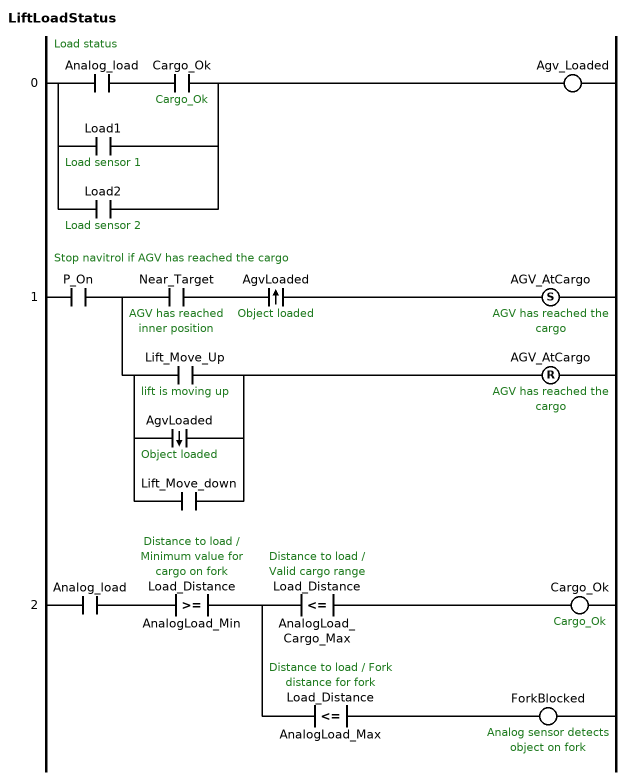
(* [picture p91: LiftLoadStatus, rungs 0-2] *)
(* Rung 0: Load status *)
Agv_Loaded := (Analog_load AND Cargo_Ok) OR Load1 OR Load2;
(* Rung 1: Stop navitrol if AGV has reached the cargo *)
_e1(CLK := AgvLoaded);
IF P_On AND Near_Target AND _e1.Q THEN AGV_AtCargo := TRUE; END_IF;
_e2(CLK := AgvLoaded);
IF P_On AND (Lift_Move_Up OR _e2.Q OR Lift_Move_down) THEN AGV_AtCargo := FALSE; END_IF;
(* Rung 2 *)
_p3 := Analog_load AND (Load_Distance >= AnalogLoad_Min);
Cargo_Ok := _p3 AND (Load_Distance <= AnalogLoad_Cargo_Max);
ForkBlocked := _p3 AND (Load_Distance <= AnalogLoad_Max);
END_FUNCTION_BLOCK

FUNCTION_BLOCK LiftAutoReset_FB
VAR
    DroppedFlag : BOOL;
END_VAR
VAR_INPUT
    Enable : BOOL;
    ControlMode : ControlLift;
    AgvLoaded : BOOL;
    Actuator_action : BOOL;
    Lift_height_actual : INT;
    Lift_height_empty : INT;
    Lift_heigt_loaded : INT;
    Dir_encoder : BOOL;
    UnloadDistance : DINT;
    M_per_rot : REAL;
    WheelEncPpr : REAL;
    ENC_position : DINT;
    ForkBlocked : BOOL;
END_VAR
VAR_OUTPUT
    ResetLift : BOOL;
    Reset_Lift_Busy : BOOL;
    Lift_Height_req_semiAuto : INT;
END_VAR
VAR_IN_OUT
    DroppedPosition : DINT;
    ResetDistance : DINT;
    ResetPosition : DINT;
END_VAR
VAR
    _e1 : F_TRIG;
    _p2 : BOOL;
    _e3 : R_TRIG;
END_VAR
(* ladder, written here as Structured Text *)

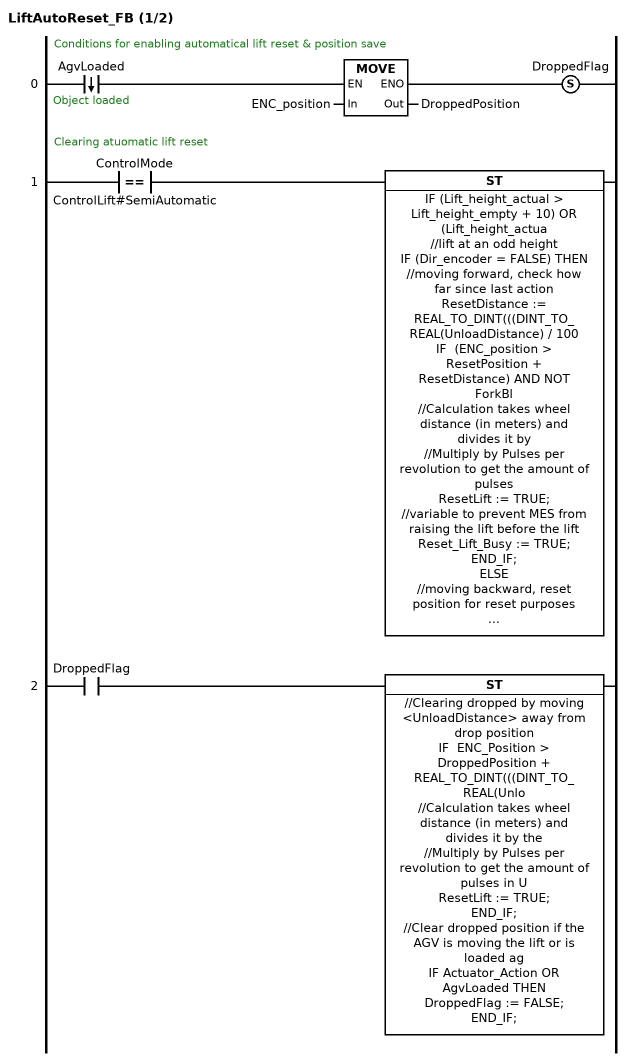
(* Rung 0: Conditions for enabling automatical lift reset & position save *)
_e1(CLK := AgvLoaded);
IF _e1.Q THEN
    DroppedPosition := ENC_position;
    DroppedFlag := TRUE;
END_IF;
(* Rung 1: Clearing atuomatic lift reset *)
IF ControlMode = ControlLift#SemiAutomatic THEN
    IF (Lift_height_actual > Lift_height_empty + 10) OR (Lift_height_actual < Lift_height_empty - 10) THEN
    	//lift at an odd height
    	IF (Dir_encoder = FALSE) THEN
    		//moving forward, check how far since last action
    		ResetDistance := REAL_TO_DINT(((DINT_TO_REAL(UnloadDistance) / 1000) / M_per_rot) * WheelEncPpr);
    		IF  (ENC_position > ResetPosition +  ResetDistance) AND NOT ForkBlocked THEN
    			//Calculation takes wheel distance (in meters) and divides it by the unload distance (in meters) to get the amount of wheel rotations in UnloadDistance. 
    			//Multiply by Pulses per revolution to get the amount of pulses in UnloadDistance.
    			ResetLift := TRUE;
    			//variable to prevent MES from raising the lift before the lift returned to normal
    			Reset_Lift_Busy := TRUE;
    		END_IF;
    	ELSE
    		//moving backward, reset position for reset purposes
    		ResetPosition := ENC_position;
    	END_IF;
    ELSE
    	//keep up with the current position
    	ResetPosition := ENC_position;
    END_IF;
END_IF;
(* Rung 2 *)
_p2 := DroppedFlag;
IF _p2 THEN
    //Clearing dropped by moving <UnloadDistance> away from drop position (and be sure fork is free)
    IF  ENC_Position > DroppedPosition +  REAL_TO_DINT(((DINT_TO_REAL(UnloadDistance) / 1000) / M_per_rot) * WheelEncPpr) AND NOT ForkBlocked THEN
    	//Calculation takes wheel distance (in meters) and divides it by the unload distance (in meters) to get the amount of wheel rotations in UnloadDistance. 
    	//Multiply by Pulses per revolution to get the amount of pulses in UnloadDistance.
    	ResetLift := TRUE;
    END_IF;
    //Clear dropped position if the AGV is moving the lift or is loaded again
    IF Actuator_Action OR AgvLoaded THEN
    	DroppedFlag := FALSE;
    END_IF;
END_IF;

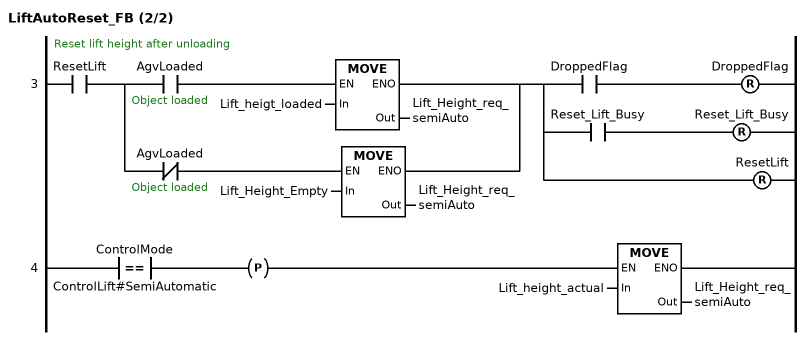
(* Rung 3: Reset lift height after unloading *)
IF ResetLift AND AgvLoaded THEN Lift_Height_req_semiAuto := Lift_heigt_loaded; END_IF;
IF ResetLift AND NOT AgvLoaded THEN Lift_Height_req_semiAuto := Lift_Height_Empty; END_IF;
IF ResetLift AND (AgvLoaded OR NOT AgvLoaded) AND DroppedFlag THEN DroppedFlag := FALSE; END_IF;
IF ResetLift AND (AgvLoaded OR NOT AgvLoaded) AND Reset_Lift_Busy THEN Reset_Lift_Busy := FALSE; END_IF;
IF ResetLift AND (AgvLoaded OR NOT AgvLoaded) THEN ResetLift := FALSE; END_IF;
(* Rung 4 *)
_e3(CLK := ControlMode = ControlLift#SemiAutomatic);
IF _e3.Q THEN Lift_Height_req_semiAuto := Lift_height_actual; END_IF;
END_FUNCTION_BLOCK

FUNCTION_BLOCK LiftCargoDrag_FB
VAR
    Difference_distance_drop : DINT;
    Difference_Pulses : REAL;
    Dropped_Flag : BOOL;
    Cargo_drag_TON : TON;
    Cargo_drag_flag : BOOL;
END_VAR
VAR_INPUT
    Enable : BOOL;
    Control_mode : ControlLift;
    Reset_flag : BOOL;
    Agv_loaded : BOOL;
    ENC_position : DINT;
    WheelEncPpr : REAL;
    M_per_Rot : REAL;
    Load_distance_real : REAL;
    Cargo_drag_PT : TIME;
END_VAR
VAR_OUTPUT
    Warning_cargo_drag : BOOL;
    Cargo_drag_ET : TIME;
END_VAR
VAR_IN_OUT
    Distance_traveled_in_m : REAL;
    Dropped_Position : DINT;
END_VAR
VAR_EXTERNAL
    AgvLoaded : BOOL;
END_VAR
VAR
    _e1 : F_TRIG;
    _e2 : R_TRIG;
END_VAR
(* ladder, written here as Structured Text *)

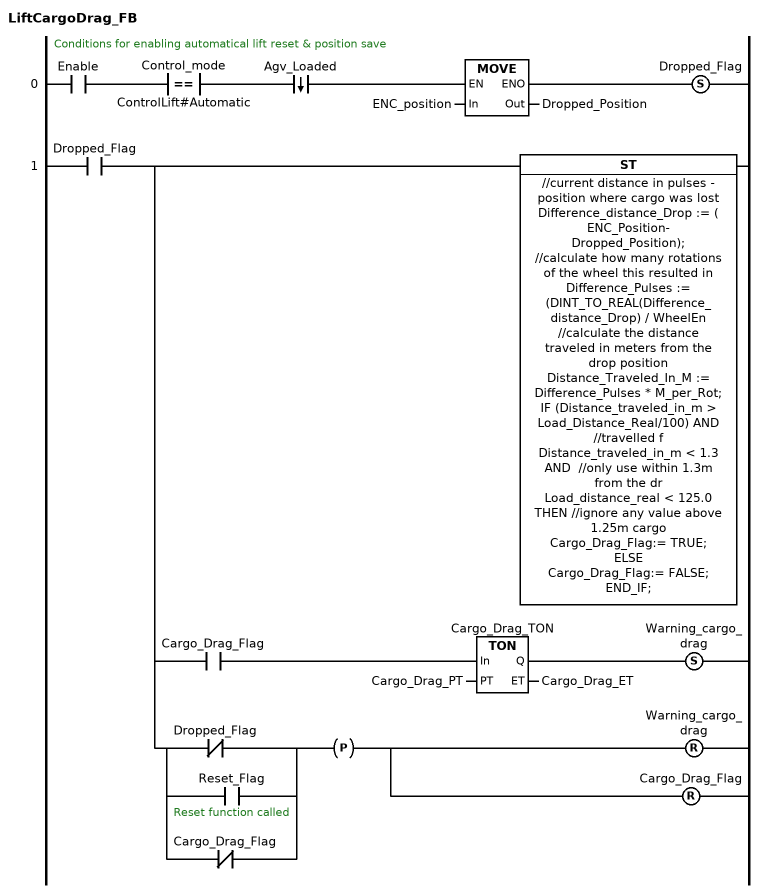
(* Rung 0: Conditions for enabling automatical lift reset & position save *)
_e1(CLK := Agv_Loaded);
IF Enable AND (Control_mode = ControlLift#Automatic) AND _e1.Q THEN
    Dropped_Position := ENC_position;
    Dropped_Flag := TRUE;
END_IF;
(* Rung 1 *)
IF Dropped_Flag THEN
    //current distance in pulses - position where cargo was lost
    Difference_distance_Drop := ( ENC_Position- Dropped_Position);
    //calculate how many rotations of the wheel this resulted in
    Difference_Pulses := (DINT_TO_REAL(Difference_distance_Drop) / WheelEncPpr);
    //calculate the distance traveled in meters from the drop position
    Distance_Traveled_In_M := Difference_Pulses * M_per_Rot;
    
    IF (Distance_traveled_in_m > Load_Distance_Real/100) AND //travelled further than the cargo?
    	Distance_traveled_in_m < 1.3 AND	//only use within 1.3m from the drop point
    	Load_distance_real < 125.0 THEN	//ignore any value above 1.25m cargo detection
    	Cargo_Drag_Flag:= TRUE;
    ELSE
    	Cargo_Drag_Flag:= FALSE;
    END_IF;
END_IF;
Cargo_Drag_TON(In := Dropped_Flag AND Cargo_Drag_Flag, PT := Cargo_Drag_PT, ET => Cargo_Drag_ET);
IF Cargo_Drag_TON.Q THEN Warning_cargo_drag := TRUE; END_IF;
_e2(CLK := Dropped_Flag AND (NOT Dropped_Flag OR Reset_Flag OR NOT Cargo_Drag_Flag));
IF _e2.Q THEN
    Warning_cargo_drag := FALSE;
    Cargo_Drag_Flag := FALSE;
END_IF;
END_FUNCTION_BLOCK

FUNCTION_BLOCK LiftHeavyLoadDetectionMax_FB
VAR_INPUT
    Enable : BOOL;
    Agv_heavy_Load_type_sensor : INT;  (* 0 = uses no sensor 1=digital sensor 2= analog sensor *)
    Heavy_weight_detection : BOOL;
    Max_weight : INT;
    Current_weight : INT;
END_VAR
VAR_OUTPUT
    Heavy_load : BOOL;
END_VAR
(* ladder, written here as Structured Text *)

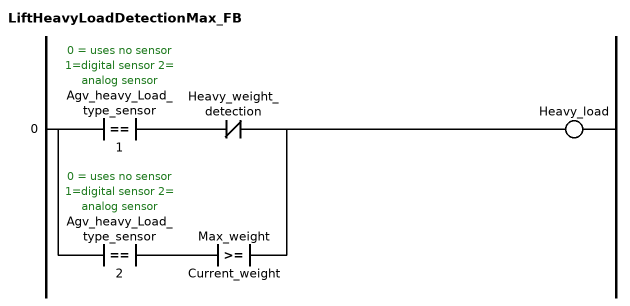
(* Rung 0 *)
Heavy_load := ((Agv_heavy_Load_type_sensor = 1) AND NOT Heavy_weight_detection) OR ((Agv_heavy_Load_type_sensor = 2) AND (Max_weight >= Current_weight));
END_FUNCTION_BLOCK

FUNCTION_BLOCK SendAckFatal
VAR
    DataReady : BOOL;  (* Data set ready for transmission *)
    TxBusy : BOOL;  (* Transmission in progress *)
    Data : Navitrol_AbortDrive_struct;
    SendDat : ARRAY[0..7] OF BYTE;  (* Data to send *)
    Messagesize : UINT;  (* Amount of bytes *)
    SendData : SktTCPSend;
END_VAR
VAR_INPUT
    Enable : BOOL;  (* Request to send *)
END_VAR
VAR_OUTPUT
    Done : BOOL;  (* Transmission done *)
END_VAR
VAR_INPUT
    Socket : _sSOCKET;  (* Navitrol socket *)
END_VAR
VAR_OUTPUT
    Error : BOOL;  (* Error during transmission *)
    ErrorID : WORD;  (* Error ID *)
END_VAR
VAR
    _e1 : R_TRIG;
    _p2 : BOOL;
    _p3 : BOOL;
    _e4 : R_TRIG;
END_VAR
(* ladder, written here as Structured Text *)

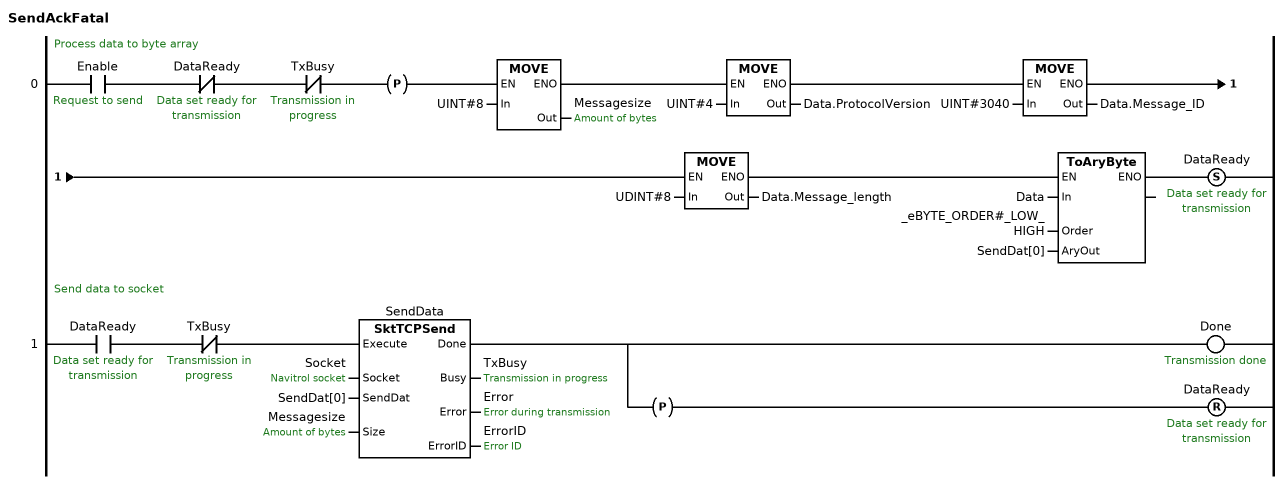
(* Rung 0: Process data to byte array *)
_e1(CLK := Enable AND NOT DataReady AND NOT TxBusy);
IF _e1.Q THEN
    Messagesize := UINT#8;
    Data.ProtocolVersion := UINT#4;
    Data.Message_ID := UINT#3040;
    Data.Message_length := UDINT#8;
    ToAryByte(In := Data, Order := _eBYTE_ORDER#_LOW_HIGH, AryOut := SendDat[0]);
    DataReady := TRUE;
END_IF;
(* Rung 1: Send data to socket *)
_p2 := DataReady AND NOT TxBusy;
SendData(Execute := _p2, Socket := Socket, SendDat := SendDat[0], Size := Messagesize, Busy => TxBusy, Error => Error, ErrorID => ErrorID);
_p3 := SendData.Done;
Done := _p3;
_e4(CLK := _p3);
IF _e4.Q THEN DataReady := FALSE; END_IF;
END_FUNCTION_BLOCK

FUNCTION_BLOCK WarningList
VAR
    WarningIndex : USINT;
END_VAR
VAR_OUTPUT
    OUT : BOOL;
END_VAR
VAR_INPUT
    IN : BOOL;
    i_BufferError : stBufferError;
    i_StoppedByOverhang : BOOL;
    ForkBlocked : BOOL;  (* Analog sensor detects object on fork *)
    Overhang_overruled : BOOL;
    FINS_enabled : BOOL;
    MES_Live : BOOL;
    StopByLowOpstacle : BOOL;
    SilentMode : BOOL;
END_VAR
VAR_EXTERNAL
    Scanner_Stop : BOOL;  (* object in safety field *)
    Warning_ActuatorTime : BOOL;  (* Lift action took too long *)
    Brake_release : BOOL;
    Manual_ControlModeLift : BOOL;
    Navitrol_status : Navitrol_Status_Struct;
    Scanner_Slowdown : BOOL;  (* object in slowdown field *)
    Scanner_Warning : BOOL;  (* object in outer field *)
    Warning_Cover_Open : BOOL;  (* One or more covers are not closed *)
    StopRequest : BOOL;
    AGV_Docking : BOOL;
    Warning_NoPallet : BOOL;  (* Cargo sensors did not detect load properly *)
    Warning_Lift_NOK : BOOL;  (* Lift sensor not in valid range *)
    Error_Navitrol : BOOL;  (* Navitrol reports an error *)
    WarningCount : USINT;  (* Amount of active warnings counter *)
    PLC_Warn_Array : array[0..4] of PLC_Warn_struct;
    Warning_TableLift_Without_load : BOOL;  (* Table has been ordered to rise without load present *)
    Warning_TableDrop_Without_Load : BOOL;  (* Table has been ordered to lower without load *)
    Warning_TableLoad_Lost : BOOL;  (* Lost tabel load while lift was high *)
    HMI_Warning1 : UINT;
    HMI_WarningText1 : INT;
    HMI_Warning2 : UINT;
    HMI_WarningText2 : INT;
    HMI_Warning3 : UINT;
    HMI_WarningText3 : INT;
    HMI_Warning4 : UINT;
    HMI_WarningText4 : INT;
    HMI_Warning5 : UINT;
    HMI_WarningText5 : INT;
    HMI_Input5 : BOOL;
    TCPReady : BOOL;
    AgvLoaded : BOOL;  (* Object loaded *)
    ClientConnected : BOOL;
    MQTT_enabled : BOOL;
    AGV_Docking_Lane : BOOL;
    HMI_Input12 : BOOL;
END_VAR
IF IN THEN		
		WarningCount := 0;

		IF AGV_Docking OR AGV_Docking_Lane then
			IF WarningCount < 5 THEN
				PLC_Warn_Array[WarningCount].WarnCode := 5101;
				PLC_Warn_Array[WarningCount].Description := 'Docking mode enabled';
				PLC_Warn_Array[WarningCount].HMI_id := 1;
				WarningCount := WarningCount + 1;
			END_IF;
		END_IF;

		IF Warning_TableLift_Without_load then
			IF WarningCount < 5 THEN
				PLC_Warn_Array[WarningCount].WarnCode := 5201;
				PLC_Warn_Array[WarningCount].Description := 'Pick without load';
				PLC_Warn_Array[WarningCount].HMI_id := 2;
				WarningCount := WarningCount + 1;
			END_IF;
		END_IF;

		IF Warning_TableDrop_Without_Load then
			IF WarningCount < 5 THEN
				PLC_Warn_Array[WarningCount].WarnCode := 5202;
				PLC_Warn_Array[WarningCount].Description := 'Drop without cargo';
				PLC_Warn_Array[WarningCount].HMI_id := 3;
				WarningCount := WarningCount + 1;
			END_IF;
		END_IF;

		IF Warning_TableLoad_Lost then
			IF WarningCount < 5 THEN
				PLC_Warn_Array[WarningCount].WarnCode := 5203;
				PLC_Warn_Array[WarningCount].Description := 'Lift has lost cargo';
				PLC_Warn_Array[WarningCount].HMI_id := 4;
				WarningCount := WarningCount + 1;
			END_IF;
		END_IF;

		IF Warning_ActuatorTime then
			IF WarningCount < 5 THEN
				PLC_Warn_Array[WarningCount].WarnCode := 5204;
				PLC_Warn_Array[WarningCount].Description := 'Actuator time exceeded';
				PLC_Warn_Array[WarningCount].HMI_id := 5;
				WarningCount := WarningCount + 1;
			END_IF;
		END_IF;

		IF MQTT_enabled AND Warning_NoPallet then
			IF WarningCount < 5 THEN
				PLC_Warn_Array[WarningCount].WarnCode := 5205;
				PLC_Warn_Array[WarningCount].Description := 'No cargo detected';
				PLC_Warn_Array[WarningCount].HMI_id := 6;
				WarningCount := WarningCount + 1;
			END_IF;
		END_IF;

		IF Warning_Lift_NOK then
			IF WarningCount < 5 THEN
				PLC_Warn_Array[WarningCount].WarnCode := 5206;
				PLC_Warn_Array[WarningCount].Description := 'Lift sensor out of range';
				PLC_Warn_Array[WarningCount].HMI_id := 7;
				WarningCount := WarningCount + 1;
			END_IF;
		END_IF;

		IF SilentMode then
			IF WarningCount < 5 THEN
				PLC_Warn_Array[WarningCount].WarnCode := 5301;
				PLC_Warn_Array[WarningCount].Description := 'Silent mode enabled';
				PLC_Warn_Array[WarningCount].HMI_id := 8;
				WarningCount := WarningCount + 1;
			END_IF;
		END_IF;

		IF Warning_Cover_Open then
			IF WarningCount < 5 THEN
				PLC_Warn_Array[WarningCount].WarnCode := 5401;
				PLC_Warn_Array[WarningCount].Description := 'Cover or door open';
				PLC_Warn_Array[WarningCount].HMI_id := 9;
				WarningCount := WarningCount + 1;
			END_IF;
		END_IF;

		IF WarningCount < 5 THEN
			IF Overhang_overruled then
				PLC_Warn_Array[WarningCount].WarnCode := 5403;
				PLC_Warn_Array[WarningCount].Description := 'Overhang overruled';
				PLC_Warn_Array[WarningCount].HMI_id := 11;
			ELSIF i_StoppedByOverhang then
				PLC_Warn_Array[WarningCount].WarnCode := 5402;
				PLC_Warn_Array[WarningCount].Description := 'Overhang detected';
				PLC_Warn_Array[WarningCount].HMI_id := 10;
			END_IF;
			WarningCount := WarningCount + 1;
		END_IF;


		IF Manual_ControlModeLift then
			IF WarningCount < 5 THEN
				PLC_Warn_Array[WarningCount].WarnCode := 5404;
				PLC_Warn_Array[WarningCount].Description := 'Manual mode active';
				PLC_Warn_Array[WarningCount].HMI_id := 12;
				WarningCount := WarningCount + 1;
			END_IF;
		END_IF;

		IF StopRequest then
			IF WarningCount < 5 THEN
				PLC_Warn_Array[WarningCount].WarnCode := 5405;
				PLC_Warn_Array[WarningCount].Description := 'Safety PLC stop request';
				PLC_Warn_Array[WarningCount].HMI_id := 13;
				WarningCount := WarningCount + 1;
			END_IF;
		END_IF;

		IF HMI_Input12 then
			IF WarningCount < 5 THEN
				PLC_Warn_Array[WarningCount].WarnCode := 5406;
				PLC_Warn_Array[WarningCount].Description := 'Operator deleted action';
				PLC_Warn_Array[WarningCount].HMI_id := 14;
				WarningCount := WarningCount + 1;
			END_IF;
		END_IF;

		IF Scanner_Warning & Scanner_Slowdown & NOT Scanner_Stop then
			IF WarningCount < 5 THEN
				PLC_Warn_Array[WarningCount].WarnCode := 5501;
				PLC_Warn_Array[WarningCount].Description := 'Object in stop field';
				PLC_Warn_Array[WarningCount].HMI_id := 15;
				WarningCount := WarningCount + 1;
			END_IF;
		END_IF;

		IF Error_Navitrol & (Navitrol_status.Pos_Conf > 30) then
			IF WarningCount < 5 THEN
				PLC_Warn_Array[WarningCount].WarnCode := 5602;
				PLC_Warn_Array[WarningCount].Description := 'Navigation in error';
				PLC_Warn_Array[WarningCount].HMI_id := 17;
				WarningCount := WarningCount + 1;
			END_IF;
		END_IF;

		IF Error_Navitrol & (Navitrol_status.Pos_Conf < 30) then
			IF WarningCount < 5 THEN
				PLC_Warn_Array[WarningCount].WarnCode := 5603;
				PLC_Warn_Array[WarningCount].Description := 'Navigation is lost';
				PLC_Warn_Array[WarningCount].HMI_id := 18;
				WarningCount := WarningCount + 1;
			END_IF;
		END_IF;

		IF p_off then
			IF WarningCount < 5 THEN
				PLC_Warn_Array[WarningCount].WarnCode := 5207;
				PLC_Warn_Array[WarningCount].Description := 'Pallet override active';
				PLC_Warn_Array[WarningCount].HMI_id := 19;
				WarningCount := WarningCount + 1;
			END_IF;
		END_IF;

		IF ForkBlocked AND NOT AgvLoaded then
			IF WarningCount < 5 THEN
				PLC_Warn_Array[WarningCount].WarnCode := 5209;
				PLC_Warn_Array[WarningCount].Description := 'Cargo location invalid';
				PLC_Warn_Array[WarningCount].HMI_id := 21;
				WarningCount := WarningCount + 1;
			END_IF;
		END_IF;

		IF Brake_release then
			IF WarningCount < 5 THEN
				PLC_Warn_Array[WarningCount].WarnCode := 5407;
				PLC_Warn_Array[WarningCount].Description := 'Brakes released';
				PLC_Warn_Array[WarningCount].HMI_id := 22;
				WarningCount := WarningCount + 1;
			END_IF;
		END_IF;

		IF HMI_Input5 then
			IF WarningCount < 5 THEN
				PLC_Warn_Array[WarningCount].WarnCode := 5408;
				PLC_Warn_Array[WarningCount].Description := 'Lift action overruled';
				PLC_Warn_Array[WarningCount].HMI_id := 23;
				WarningCount := WarningCount + 1;
			END_IF;
		END_IF;

		//communication warnings
		IF (NOT TCPReady) THEN
			IF WarningCount < 5 THEN
				PLC_Warn_Array[WarningCount].WarnCode := 5701;
				PLC_Warn_Array[WarningCount].Description := 'Navitrol offline';
				PLC_Warn_Array[WarningCount].HMI_id := 24;
				WarningCount := WarningCount + 1;
			END_IF;
		END_IF;

		IF (FINS_enabled AND NOT MES_Live) THEN
			IF WarningCount < 5 THEN
				PLC_Warn_Array[WarningCount].WarnCode := 5702;
				PLC_Warn_Array[WarningCount].Description := 'FINS timeout to MES';
				PLC_Warn_Array[WarningCount].HMI_id := 25;
				WarningCount := WarningCount + 1;
			END_IF;
		END_IF;

		IF (MQTT_enabled AND NOT ClientConnected) THEN
			IF WarningCount < 5 THEN
				PLC_Warn_Array[WarningCount].WarnCode := 5703;
				PLC_Warn_Array[WarningCount].Description := 'Mqtt broker offline';
				PLC_Warn_Array[WarningCount].HMI_id := 26;
				WarningCount := WarningCount + 1;
			END_IF;
		END_IF;

		(*IF  then
			IF WarningCount < 5 THEN
				PLC_Warn_Array[WarningCount].WarnCode := 5405;
				PLC_Warn_Array[WarningCount].Description := 'AGV in stopzone';
				PLC_Warn_Array[WarningCount].HMI_id := 27;
				WarningCount := WarningCount + 1;
			END_IF;
		END_IF;

		IF  then
			IF WarningCount < 5 THEN
				PLC_Warn_Array[WarningCount].WarnCode := 5210;
				PLC_Warn_Array[WarningCount].Description := 'Pallet stack height detection active';
				PLC_Warn_Array[WarningCount].HMI_id := 28;
				WarningCount := WarningCount + 1;
			END_IF;
		END_IF;

		IF  then
			IF WarningCount < 5 THEN
				PLC_Warn_Array[WarningCount].WarnCode := 5211;
				PLC_Warn_Array[WarningCount].Description := 'Too many pallets detect.';
				PLC_Warn_Array[WarningCount].HMI_id := 29;
				WarningCount := WarningCount + 1;
			END_IF;
		END_IF;
		*)

		IF StopByLowOpstacle then
			IF WarningCount < 5 THEN
				PLC_Warn_Array[WarningCount].WarnCode := 5409;
				PLC_Warn_Array[WarningCount].Description := 'Low sensor detec object';
				PLC_Warn_Array[WarningCount].HMI_id := 30;
				WarningCount := WarningCount + 1;
			END_IF;
		END_IF;
		
		IF P_Off THEN
			IF WarningCount < 5 THEN
				PLC_Warn_Array[WarningCount].WarnCode := 5411;
				PLC_Warn_Array[WarningCount].Description := 'Lane sensor out of range';
				PLC_Warn_Array[WarningCount].HMI_id := 31;
				WarningCount := WarningCount + 1;
			END_IF;
		END_IF;

		IF i_BufferError.LiftHeight THEN
			IF WarningCount < 5 THEN
				PLC_Warn_Array[WarningCount].WarnCode := 5412;
				PLC_Warn_Array[WarningCount].Description := 'Too low lift height lane';
				PLC_Warn_Array[WarningCount].HMI_id := 32;
				WarningCount := WarningCount + 1;
			END_IF;
		END_IF;
		
		IF i_BufferError.CargoSensorBWIRE THEN
			IF WarningCount < 5 THEN
				PLC_Warn_Array[WarningCount].WarnCode := 5413;
				PLC_Warn_Array[WarningCount].Description := 'Cargo sensor broke wire';
				PLC_Warn_Array[WarningCount].HMI_id := 33;
				WarningCount := WarningCount + 1;
			END_IF;
		END_IF;

		IF (WarningCount < 5) THEN
			PLC_Warn_Array[4].WarnCode := 0;
			PLC_Warn_Array[4].Description := '                        ';
			PLC_Warn_Array[4].HMI_id := 0;
		END_IF;
		IF (WarningCount < 4) THEN
			PLC_Warn_Array[3].WarnCode := 0;
			PLC_Warn_Array[3].Description := '                        ';
			PLC_Warn_Array[3].HMI_id := 0;
		END_IF;
		IF (WarningCount < 3) THEN
			PLC_Warn_Array[2].WarnCode := 0;
			PLC_Warn_Array[2].Description := '                        ';
			PLC_Warn_Array[2].HMI_id := 0;
		END_IF;
		IF (WarningCount < 2) THEN
			PLC_Warn_Array[1].WarnCode := 0;
			PLC_Warn_Array[1].Description := '                        ';
			PLC_Warn_Array[1].HMI_id := 0;
		END_IF;
		IF (WarningCount < 1) THEN
			//no warnings active
			PLC_Warn_Array[0].WarnCode := 0;
			PLC_Warn_Array[0].Description := '                        ';
			PLC_Warn_Array[0].HMI_id := 0;
		END_IF;

		//Handle the error strings
		FOR WarningIndex := 0 to 4 DO
			PLC_Warn_Array[WarningIndex].ActualChars := uint_to_byte(LEN(PLC_Warn_Array[WarningIndex].Description));
			PLC_Warn_Array[WarningIndex].ZeroFill := int_to_byte(BYTE_TO_INT(PLC_Warn_Array[WarningIndex].DescrLength) -BYTE_TO_INT(PLC_Warn_Array[WarningIndex].ActualChars));
		END_FOR;

		//HMI_WarningText1 := '                        ';
		//HMI_WarningText2 := '                        ';
		//HMI_WarningText3 := '                        ';
		//HMI_WarningText4 := '                        ';
		//HMI_WarningText5 := '                        ';

		HMI_Warning1 := PLC_Warn_Array[0].WarnCode;
		HMI_WarningText1 := BYTE_TO_INT(PLC_Warn_Array[0].HMI_id);
		HMI_Warning2 := PLC_Warn_Array[1].WarnCode;
		HMI_WarningText2 :=  BYTE_TO_INT(PLC_Warn_Array[1].HMI_id);
		HMI_Warning3 := PLC_Warn_Array[2].WarnCode;
		HMI_WarningText3 :=  BYTE_TO_INT(PLC_Warn_Array[2].HMI_id);
		HMI_Warning4 := PLC_Warn_Array[3].WarnCode;
		HMI_WarningText4 :=  BYTE_TO_INT(PLC_Warn_Array[3].HMI_id);
		HMI_Warning5 := PLC_Warn_Array[4].WarnCode;
		HMI_WarningText5 :=  BYTE_TO_INT(PLC_Warn_Array[4].HMI_id);
END_IF;
END_FUNCTION_BLOCK

FUNCTION_BLOCK Bufferlane_FB
VAR
    STANDSTILL_CARGO_DIST_MIN : REAL := 970;  (* Minimum value cargo should be *)
    DistSensor : stAnalogSensor;
    LoadSwitchDelay1 : TOF;
    NAVITROL_BUFFERLANE_FIRST : REAL := 1;  (* AGV in bufferlane *)
    BUFFERLANE_PICK : INT := 1;  (* MES defined action 1 *)
    BUFFERLANE_DROP : INT := 2;  (* MES defined action 2 *)
    BUFFERLANE_DROP_HEIGHT : INT := 295;  (* Drop height in bufferlane, customer Alpma *)
    HoldOnPosition : BOOL;  (* Keep AGV on position *)
    BUFFERLANE_PICK_HEIGHT : INT := 460;  (* Pick height in bufferlane, customer Alpma *)
    PICKING_ACTION : INT := 40;  (* Enum values picking *)
    DROPPING_ACTION : INT := 40;  (* Enum values dropping *)
    TARGET_REACHED : UINT := 1;
    ENTER_LANE_LIFT_MARGE : INT := 10;
    NAVITROL_BUFFERLANE_OUT : REAL := 4;
    DIST_TO_TARGET_MIN : REAL := 0.2;  (* AGV does stop at target instead sensor *)
    SP_SLOW : INT;
    SP_STOP : INT;
    ANALOG_LANE_SENSOR : INT := 1;  (* Analog sensor to stop AGV *)
END_VAR
VAR_INPUT
    ENABLE : BOOL;
    CNTRL : stControl;
    i_LaneStateMES : Lane_state_MES;
    i_SensorType : INT;
    i_BufferLaneSensorDistance : INT;
    i_Load_Distance : REAL;
    i_LiftReqAuto : INT;
    i_ClampSTS : BOOL;
    i_Lift_Height : INT;  (* Calculated lift height *)
    i_ReadyToClamp : BOOL;  (* Calculated lift height *)
    i_Lift_Mode : ControlLift;  (* Lift control mode *)
END_VAR
VAR_OUTPUT
    STOP_POS : BOOL;  (* AGV stopped by used distance and cargo sensor *)
    SPD_LIM : BOOL;  (* AGV gets limited in speed *)
    STATUS : stBufferlaneStatus;
    ErrType : stBufferError;
    ERROR : BOOL;
END_VAR
VAR_EXTERNAL
    Load_Distance : INT;
    Manual_Navitrol : BOOL;
    Navitrol_ProductionStatus : Navitrol_ProductionData_struct;
    Navitrol_DriveInfo : Navitrol_Status_DriveorderInfo_sec_struct;
    Navitrol_DistanceInfo : Navitrol_Status_DistanceToTarget_sec_struct;
    Standstill : BOOL;
    ClampAttached : BOOL;
    Scan3_Stop : BOOL;
    Scan3_Warn : BOOL;
    ActuatorAction : BOOL;
    RequestDriveReady : BOOL;
END_VAR
VAR
    _e1 : F_TRIG;
    _e2 : F_TRIG;
    _e3 : R_TRIG;
    _e4 : R_TRIG;
    _e5 : R_TRIG;
    _e6 : R_TRIG;
    _e7 : R_TRIG;
    _e8 : R_TRIG;
    _e9 : F_TRIG;
END_VAR
(* ladder, written here as Structured Text *)

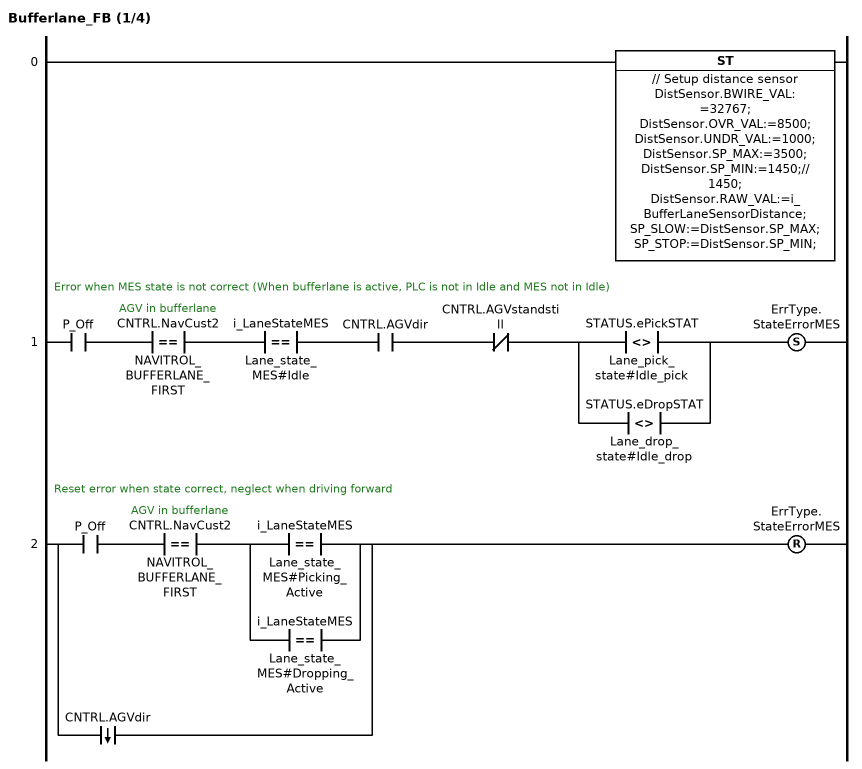
(* Rung 0 *)
// Setup distance sensor

DistSensor.BWIRE_VAL:=32767;
DistSensor.OVR_VAL:=8500;
DistSensor.UNDR_VAL:=1000;
DistSensor.SP_MAX:=3500;
DistSensor.SP_MIN:=1450;//1450;
DistSensor.RAW_VAL:=i_BufferLaneSensorDistance;

SP_SLOW:=DistSensor.SP_MAX;
SP_STOP:=DistSensor.SP_MIN;
(* Rung 1: Error when MES state is not correct (When bufferlane is active, PLC is not in Idle and MES not in Idle) *)
IF P_Off AND (CNTRL.NavCust2 = NAVITROL_BUFFERLANE_FIRST) AND (i_LaneStateMES = Lane_state_MES#Idle) AND CNTRL.AGVdir AND NOT CNTRL.AGVstandstill AND ((STATUS.ePickSTAT <> Lane_pick_state#Idle_pick) OR (STATUS.eDropSTAT <> Lane_drop_state#Idle_drop)) THEN
    ErrType.StateErrorMES := TRUE;
END_IF;
(* Rung 2: Reset error when state correct, neglect when driving forward *)
_e1(CLK := CNTRL.AGVdir);
IF (P_Off AND (CNTRL.NavCust2 = NAVITROL_BUFFERLANE_FIRST) AND ((i_LaneStateMES = Lane_state_MES#Picking_Active) OR (i_LaneStateMES = Lane_state_MES#Dropping_Active))) OR _e1.Q THEN
    ErrType.StateErrorMES := FALSE;
END_IF;

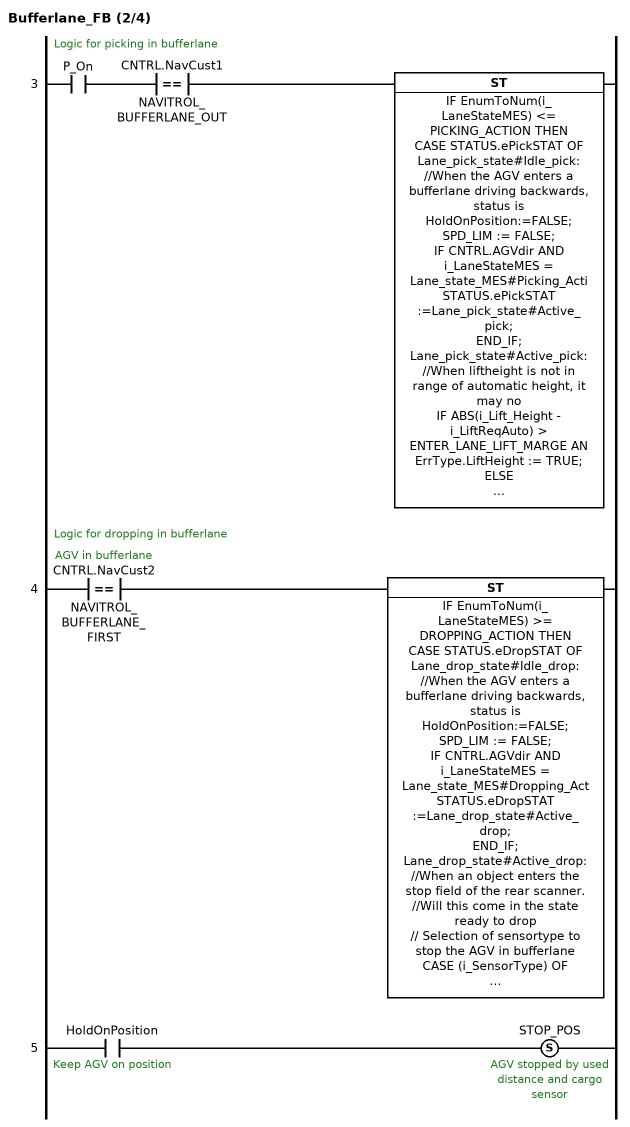
(* Rung 3: Logic for picking in bufferlane *)
IF P_On AND (CNTRL.NavCust1 = NAVITROL_BUFFERLANE_OUT) THEN
    IF EnumToNum(i_LaneStateMES) <= PICKING_ACTION THEN	
    	CASE STATUS.ePickSTAT OF
    		Lane_pick_state#Idle_pick:
    			//When the AGV enters a bufferlane driving backwards, status is active pick
    			HoldOnPosition:=FALSE;
    			SPD_LIM := FALSE;
    			IF CNTRL.AGVdir AND i_LaneStateMES = Lane_state_MES#Picking_Active THEN 
    				STATUS.ePickSTAT :=Lane_pick_state#Active_pick;
    			END_IF;
    
    		Lane_pick_state#Active_pick:
    			//When liftheight is not in range of automatic height, it may not drive automatically in lane!
    			IF ABS(i_Lift_Height - i_LiftReqAuto) > ENTER_LANE_LIFT_MARGE AND CNTRL.AGVdir AND CNTRL.NavInProduction  = 1 THEN
    				ErrType.LiftHeight := TRUE;
    			ELSE
    				ErrType.LiftHeight := FALSE;
    			END_IF;
    			
    			// Selection of sensortype to stop the AGV in bufferlane
    			CASE (i_SensorType) OF
    				1:
    					//Analog has max setpoint for slowdown and min setpoint for stopping AGV
    					IF DistSensor.RAW_VAL < SP_SLOW THEN
    						SPD_LIM := TRUE;
    					END_IF;
    					IF DistSensor.RAW_VAL < SP_STOP AND CNTRL.AGVdir THEN
    						HoldOnPosition := TRUE;
    						IF CNTRL.AGVstandstill AND i_LaneStateMES = Lane_state_MES#Picking_Active THEN
    							STATUS.ePickSTAT := Ready_to_lower_lift_pick;
    						END_IF;
    					END_IF;
    				
    				//AGV stopts already when safety scanner sees an object in stopfield
    				2:
    					IF Scan3_Stop THEN
    						IF CNTRL.AGVstandstill AND i_LaneStateMES = Lane_state_MES#Picking_Active THEN
    							STATUS.ePickSTAT := Ready_to_lower_lift_pick;
    						END_IF;
    					END_IF;				
    			END_CASE;
    			
    		
    		Lane_pick_state#Ready_to_lower_lift_pick:
    			// HoldOnPosition while lowering lift
    			HoldOnPosition := ActuatorAction;
    		
    			//When the lift is lowered, AGV can drive with forks under load
    			IF i_LaneStateMES = Lane_state_MES#Picking_Drive_In THEN
    				HoldOnPosition := FALSE;
    			END_IF;
    			//AGV does not stop on cargo sensor, but symbolic point if distance is less than DIST_TO_TARGET_MIN
    			IF Navitrol_DistanceInfo.DistanceToTarget <= DIST_TO_TARGET_MIN THEN
    				IF NOT i_ReadyToClamp AND CNTRL.AGVstandstill THEN
    					STATUS.ePickSTAT := Ready_to_pick;
    				END_IF;
    			ELSE
    			//Otherwise AGV stops when it is loaded
    				IF CNTRL.AGVloaded THEN
    					HoldOnPosition:=TRUE;
    					IF NOT i_ReadyToClamp AND CNTRL.AGVstandstill THEN
    						STATUS.ePickSTAT := Ready_to_pick;
    					END_IF;
    				END_IF;
    			END_IF;
    			
    		Lane_pick_state#Ready_to_pick:
    			//When the AGV has picked the cargo, it will be reversed by the MES application.
    			//From that moment on, the state is changed to idle.
    			IF i_LaneStateMES = Lane_state_MES#Picking_Finished THEN
    				IF ClampAttached AND i_ClampSTS THEN
    					STATUS.ePickSTAT := Idle_pick;
    				ELSIF NOT ClampAttached THEN
    					STATUS.ePickSTAT := Idle_pick;
    				END_IF;
    			END_IF;
    	END_CASE;
    
    	//When the AGV drives out the lane-picking lane, the lanepick state is written to idle.
    	IF NOT CNTRL.AGVdir AND NOT CNTRL.AGVstandstill THEN
    		STATUS.ePickSTAT := Idle_pick;
    	END_IF;
    END_IF;
END_IF;
(* Rung 4: Logic for dropping in bufferlane *)
IF CNTRL.NavCust2 = NAVITROL_BUFFERLANE_FIRST THEN
    IF EnumToNum(i_LaneStateMES) >= DROPPING_ACTION THEN	
    	CASE STATUS.eDropSTAT OF
    		Lane_drop_state#Idle_drop:
    			//When the AGV enters a bufferlane driving backwards, status is active drop
    			HoldOnPosition:=FALSE;
    			SPD_LIM := FALSE;
    			IF CNTRL.AGVdir AND i_LaneStateMES = Lane_state_MES#Dropping_Active THEN
    				STATUS.eDropSTAT :=Lane_drop_state#Active_drop;
    			END_IF;
    
    		Lane_drop_state#Active_drop:
    			//When an object enters the stop field of the rear scanner.
    			//Will this come in the state ready to drop	
    			
    			// Selection of sensortype to stop the AGV in bufferlane
    			CASE (i_SensorType) OF
    				1:
    					//Analog has max setpoint for slowdown and min setpoint for stopping AGV
    					IF DistSensor.RAW_VAL < SP_SLOW AND DistSensor.RAW_VAL > SP_STOP THEN
    						SPD_LIM := TRUE;
    					END_IF;
    					IF DistSensor.RAW_VAL < SP_STOP AND DistSensor.RAW_VAL > DistSensor.UNDR_VAL AND CNTRL.AGVdir  THEN
    						HoldOnPosition:=TRUE;
    						IF CNTRL.AGVstandstill AND i_LaneStateMES = Lane_state_MES#Dropping_Active THEN
    							STATUS.eDropSTAT := Ready_to_drop;
    						END_IF;	
    					END_IF;	
    				2:
    					//AGV stopts already when safety scanner sees an object in stopfield
    					IF Scan3_Stop AND Standstill THEN						 
    						IF CNTRL.AGVstandstill AND i_LaneStateMES = Lane_state_MES#Dropping_Active THEN
    							STATUS.eDropSTAT := Ready_to_drop;
    						END_IF;
    					END_IF;
    			END_CASE;
    			
    			IF i_LaneStateMES = Lane_state_MES#Dropping THEN
    					STATUS.eDropSTAT := Ready_to_drop;
    			END_IF;
    
    		Lane_drop_state#Ready_to_drop:
    			//When the AGV has dropped the pallet, it will be reversed by the MES application.
    			//And when the AGV has moved backwards enough, the lift is sent upwards.
    			//From that moment on, the state is changed to finshed.	
    			
    			// HoldOnPosition while lowering lift
    			HoldOnPosition := ActuatorAction;
    			RequestDriveReady:=TRUE;
    			
    			IF CNTRL.AGVstandstill AND i_LaneStateMES = Lane_state_MES#Dropping_Finished THEN
    				STATUS.eDropSTAT := Idle_drop;
    			END_IF;
    	END_CASE;
    
    	//When the agv is not in a lane-dropping lane.
    	//The lanedrop state is written to idle.
    	IF NOT CNTRL.AGVdir AND NOT CNTRL.AGVstandstill THEN
    		STATUS.eDropSTAT := Idle_drop;
    	END_IF;
    END_IF;
END_IF;
(* Rung 5 *)
IF HoldOnPosition THEN STOP_POS := TRUE; END_IF;

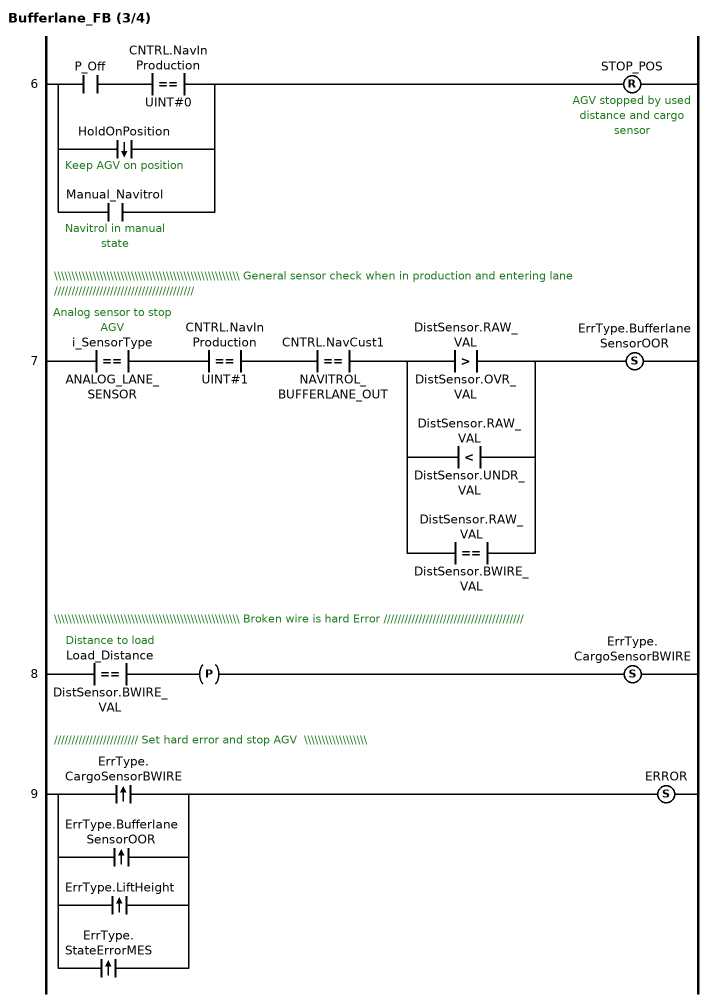
(* Rung 6 *)
_e2(CLK := HoldOnPosition);
IF (P_Off AND (CNTRL.NavInProduction = UINT#0)) OR _e2.Q OR Manual_Navitrol THEN
    STOP_POS := FALSE;
END_IF;
(* Rung 7: \\\\\\\\\\\\\\\\\\\\\\\\\\\\\\\\\\\\\\\\\\\\\\\\\\\\\ General sensor check when in production and entering lane //////////////////////////////////////// *)
IF (i_SensorType = ANALOG_LANE_SENSOR) AND (CNTRL.NavInProduction = UINT#1) AND (CNTRL.NavCust1 = NAVITROL_BUFFERLANE_OUT) AND ((DistSensor.RAW_VAL > DistSensor.OVR_VAL) OR (DistSensor.RAW_VAL < DistSensor.UNDR_VAL) OR (DistSensor.RAW_VAL = DistSensor.BWIRE_VAL)) THEN
    ErrType.BufferlaneSensorOOR := TRUE;
END_IF;
(* Rung 8: \\\\\\\\\\\\\\\\\\\\\\\\\\\\\\\\\\\\\\\\\\\\\\\\\\\\\ Broken wire is hard Error //////////////////////////////////////// *)
_e3(CLK := Load_Distance = DistSensor.BWIRE_VAL);
IF _e3.Q THEN ErrType.CargoSensorBWIRE := TRUE; END_IF;
(* Rung 9: //////////////////////// Set hard error and stop AGV  \\\\\\\\\\\\\\\\\\ *)
_e4(CLK := ErrType.CargoSensorBWIRE);
_e5(CLK := ErrType.BufferlaneSensorOOR);
_e6(CLK := ErrType.LiftHeight);
_e7(CLK := ErrType.StateErrorMES);
IF _e4.Q OR _e5.Q OR _e6.Q OR _e7.Q THEN ERROR := TRUE; END_IF;

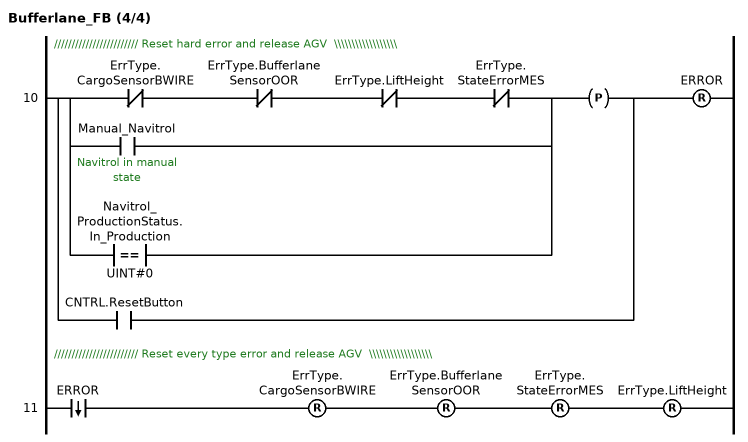
(* Rung 10: //////////////////////// Reset hard error and release AGV  \\\\\\\\\\\\\\\\\\ *)
_e8(CLK := (NOT ErrType.CargoSensorBWIRE AND NOT ErrType.BufferlaneSensorOOR AND NOT ErrType.LiftHeight AND NOT ErrType.StateErrorMES) OR Manual_Navitrol OR (Navitrol_ProductionStatus.In_Production = UINT#0));
IF _e8.Q OR CNTRL.ResetButton THEN ERROR := FALSE; END_IF;
(* Rung 11: //////////////////////// Reset every type error and release AGV  \\\\\\\\\\\\\\\\\\ *)
_e9(CLK := ERROR);
IF _e9.Q THEN
    ErrType.CargoSensorBWIRE := FALSE;
    ErrType.BufferlaneSensorOOR := FALSE;
    ErrType.StateErrorMES := FALSE;
    ErrType.LiftHeight := FALSE;
END_IF;
END_FUNCTION_BLOCK

FUNCTION_BLOCK ErrorList_FB
VAR_INPUT
    IN : BOOL;
END_VAR
VAR_OUTPUT
    OUT : BOOL;
END_VAR
VAR_EXTERNAL
    ErrorCount : USINT;
    Motor_Ok : BOOL;
    PLC_Error_Array : array[0..4] of PLC_Error_struct;
    Estop_Channel1 : BOOL;
    Error_Fork_Object : BOOL;
    Docking_error : BOOL;
    SpeedError : BOOL;
    Pump_Ok : BOOL;
    Estop_Out : BOOL;
    Scanner_Warning : BOOL;
    Scanner_Slowdown : BOOL;
    Scanner_Stop : BOOL;
    ErrorIndex : USINT;
    HMI_Error1 : UINT;
    HMI_ErrorText1 : INT;
    HMI_Error2 : UINT;
    HMI_ErrorText2 : INT;
    HMI_Error3 : UINT;
    HMI_ErrorText3 : INT;
    HMI_Error4 : UINT;
    HMI_ErrorText4 : INT;
    HMI_Error5 : UINT;
    HMI_ErrorText5 : INT;
    ENC1_Dir : BOOL;
END_VAR
IF IN THEN		
	ErrorCount := 0;

	IF (not Motor_Ok) AND Estop_Channel1 AND (NOT Error_Fork_Object) AND (NOT Docking_error) then
		IF ErrorCount < 5 THEN
			PLC_Error_Array[ErrorCount].ErrCode := 1101;
			PLC_Error_Array[ErrorCount].Description := 'Motor power not OK';
			PLC_Error_Array[ErrorCount].HMI_id := 1;
			ErrorCount := ErrorCount + 1;
		END_IF;
	END_IF;

	IF SpeedError then
		IF ErrorCount < 5 THEN
			PLC_Error_Array[ErrorCount].ErrCode := 1102;
			PLC_Error_Array[ErrorCount].Description := 'Speed check invalid';
			PLC_Error_Array[ErrorCount].HMI_id := 2;
			ErrorCount := ErrorCount + 1;
		END_IF;
	END_IF;

	IF (not Pump_Ok) AND Estop_Out AND (NOT Error_Fork_Object) then
		IF ErrorCount < 5 THEN
			PLC_Error_Array[ErrorCount].ErrCode := 1201;
			PLC_Error_Array[ErrorCount].Description := 'Lift power not OK';
			PLC_Error_Array[ErrorCount].HMI_id := 3;
			ErrorCount := ErrorCount + 1;
		END_IF;
	END_IF;
	(*
	IF heavyLoad.Q1 THEN
		IF ErrorCount < 5 THEN
			PLC_Error_Array[ErrorCount].ErrCode := 1202;
			PLC_Error_Array[ErrorCount].Description := 'Heavy load, max hight';
			PLC_Error_Array[ErrorCount].HMI_id := 15;
			ErrorCount := ErrorCount + 1;
		END_IF;
	END_IF;
	*)
	//IF Error_Navitrol then
	//	IF ErrorCount < 5 THEN
	//		PLC_Error_Array[ErrorCount].ErrCode := 1301;
	//		PLC_Error_Array[ErrorCount].Description := 'ERR_NAVITROL_TO_PLC';
	//		ErrorCount := ErrorCount + 1;
	//	END_IF;
	//END_IF;

	IF (NOT Estop_Channel1 & NOT Estop_Out) THEN
		IF ErrorCount < 5 THEN
			PLC_Error_Array[ErrorCount].ErrCode := 1401;
			PLC_Error_Array[ErrorCount].Description := 'E-stop button pressed';
			PLC_Error_Array[ErrorCount].HMI_id := 4;
			ErrorCount := ErrorCount + 1;
		END_IF;
	END_IF;

	IF (Estop_Channel1 & NOT Estop_Out) THEN
		IF ErrorCount < 5 THEN
			PLC_Error_Array[ErrorCount].ErrCode := 1402;
			PLC_Error_Array[ErrorCount].Description := 'E-stop reset required';
			PLC_Error_Array[ErrorCount].HMI_id := 5;
			ErrorCount := ErrorCount + 1;
		END_IF;
	END_IF;

	IF (Scanner_Warning & Scanner_Slowdown & Scanner_Stop) THEN
		IF ErrorCount < 5 THEN
			PLC_Error_Array[ErrorCount].ErrCode := 1403;
			PLC_Error_Array[ErrorCount].Description := 'Object in safety field';
			PLC_Error_Array[ErrorCount].HMI_id := 6;
			ErrorCount := ErrorCount + 1;
		END_IF;
	END_IF;

	IF (NOT Scanner_Warning & NOT Scanner_Slowdown & Scanner_Stop) THEN
		IF ErrorCount < 5 THEN
			PLC_Error_Array[ErrorCount].ErrCode := 1404;
			PLC_Error_Array[ErrorCount].Description := 'Scanner in fault';
			PLC_Error_Array[ErrorCount].HMI_id := 7;
			ErrorCount := ErrorCount + 1;
		END_IF;
	END_IF;

	IF (Error_Fork_Object) THEN
		IF ErrorCount < 5 THEN
			PLC_Error_Array[ErrorCount].ErrCode := 1502;
			PLC_Error_Array[ErrorCount].Description := 'Fork collision';
			PLC_Error_Array[ErrorCount].HMI_id := 8;
			ErrorCount := ErrorCount + 1;
		END_IF;
	END_IF;

	IF (Docking_error) THEN
		IF ErrorCount < 5 THEN
			PLC_Error_Array[ErrorCount].ErrCode := 1503;
			PLC_Error_Array[ErrorCount].Description := 'Docking error lane drop';
			PLC_Error_Array[ErrorCount].HMI_id := 9;
			ErrorCount := ErrorCount + 1;
		END_IF;
	END_IF;



	IF (ErrorCount < 5) THEN
		PLC_Error_Array[4].ErrCode := 0;
		PLC_Error_Array[4].Description := '                        ';
		PLC_Error_Array[4].HMI_id := 0;
	END_IF;
	IF (ErrorCount < 4) THEN
		PLC_Error_Array[3].ErrCode := 0;
		PLC_Error_Array[3].Description := '                        ';
		PLC_Error_Array[3].HMI_id := 0;
	END_IF;
	IF (ErrorCount < 3) THEN
		PLC_Error_Array[2].ErrCode := 0;
		PLC_Error_Array[2].Description := '                        ';
		PLC_Error_Array[2].HMI_id := 0;
	END_IF;
	IF (ErrorCount < 2) THEN
		PLC_Error_Array[1].ErrCode := 0;
		PLC_Error_Array[1].Description := '                        ';
		PLC_Error_Array[1].HMI_id := 0;
	END_IF;
	IF (ErrorCount < 1) THEN
		//No active errors
		PLC_Error_Array[0].ErrCode := 0;
		PLC_Error_Array[0].Description := '                        ';
		PLC_Error_Array[0].HMI_id := 0;
	END_IF;

	//Handle the error strings
	FOR ErrorIndex := 0 to 4 DO
		PLC_Error_Array[ErrorIndex].ActualChars := uint_to_byte(LEN(PLC_Error_Array[ErrorIndex].Description));
		PLC_Error_Array[ErrorIndex].ZeroFill := int_to_byte(BYTE_TO_INT(PLC_Error_Array[ErrorIndex].DescrLength) -BYTE_TO_INT(PLC_Error_Array[ErrorIndex].ActualChars));
	END_FOR;

	//HMI_ErrorText1 := '                        ';
	//HMI_ErrorText2 := '                        ';
	//HMI_ErrorText3 := '                        ';
	//HMI_ErrorText4 := '                        ';
	//HMI_ErrorText5 := '                        ';

	HMI_Error1 := PLC_Error_Array[0].ErrCode;
	HMI_ErrorText1 := BYTE_TO_INT(PLC_Error_Array[0].HMI_id);
	HMI_Error2 := PLC_Error_Array[1].ErrCode;
	HMI_ErrorText2 := BYTE_TO_INT(PLC_Error_Array[1].HMI_id);
	HMI_Error3 := PLC_Error_Array[2].ErrCode;
	HMI_ErrorText3 := BYTE_TO_INT(PLC_Error_Array[2].HMI_id);
	HMI_Error4 := PLC_Error_Array[3].ErrCode;
	HMI_ErrorText4 := BYTE_TO_INT(PLC_Error_Array[3].HMI_id);
	HMI_Error5 := PLC_Error_Array[4].ErrCode;
	HMI_ErrorText5 := BYTE_TO_INT(PLC_Error_Array[4].HMI_id);
	
END_IF;
END_FUNCTION_BLOCK

FUNCTION_BLOCK LowObstacleDET_FB
VAR
    NAVITROL_DSBL_LOW_SENSOR : REAL := 1;
    NAVITROL_ENBL_LOW_SENSOR : REAL := 0;
    Disable_Overhang : BOOL;
    UseLowObstacleDet : BOOL;
    LowOpstacleDetected : BOOL;
    i_LowObstaclesSIGNAL : BOOL;
    SetLowObstacle_TON : TON;
    LowObstacle_PT : TIME := T#250ms;
    Overhang_ET : TIME;
    Reset_Overhang_PT : TIME := T#1s;
    Overhang_ChargerOverride : BOOL;
    Disable_LowObstacleDetection : BOOL;
    LowObstacle_ChargerOverride : BOOL;
    Reset_LowObstacle_TON : TON;
    Reset_Overhang_ET : TIME;
END_VAR
VAR_INPUT
    ENABLE : BOOL;
    CNTRL : stControl;
    i_DockingActive : BOOL;
    i_LaneFieldActive : BOOL;
    i_LaneDockingActive : BOOL;
    i_UseLowObstacleDet : BOOL;
    i_LowObstacleIO : BOOL;
    i_LiftMode : ControlLift;
END_VAR
VAR_OUTPUT
    STOP : BOOL;
    ERROR : BOOL;
END_VAR
VAR_EXTERNAL
    Brake_Override_Switch : BOOL;
    Charge_Relay : BOOL;
    Navitrol_Tag : Navitrol_Status_TagV4_sec_struct;
    ToChargerTag : UDINT;
    ChargerTag : UDINT;
END_VAR
VAR
    _e1 : R_TRIG;
    _e2 : R_TRIG;
    _e3 : R_TRIG;
    _p4 : BOOL;
    _e5 : R_TRIG;
    _e6 : R_TRIG;
    _e7 : R_TRIG;
    _e8 : R_TRIG;
END_VAR
(* ladder, written here as Structured Text *)

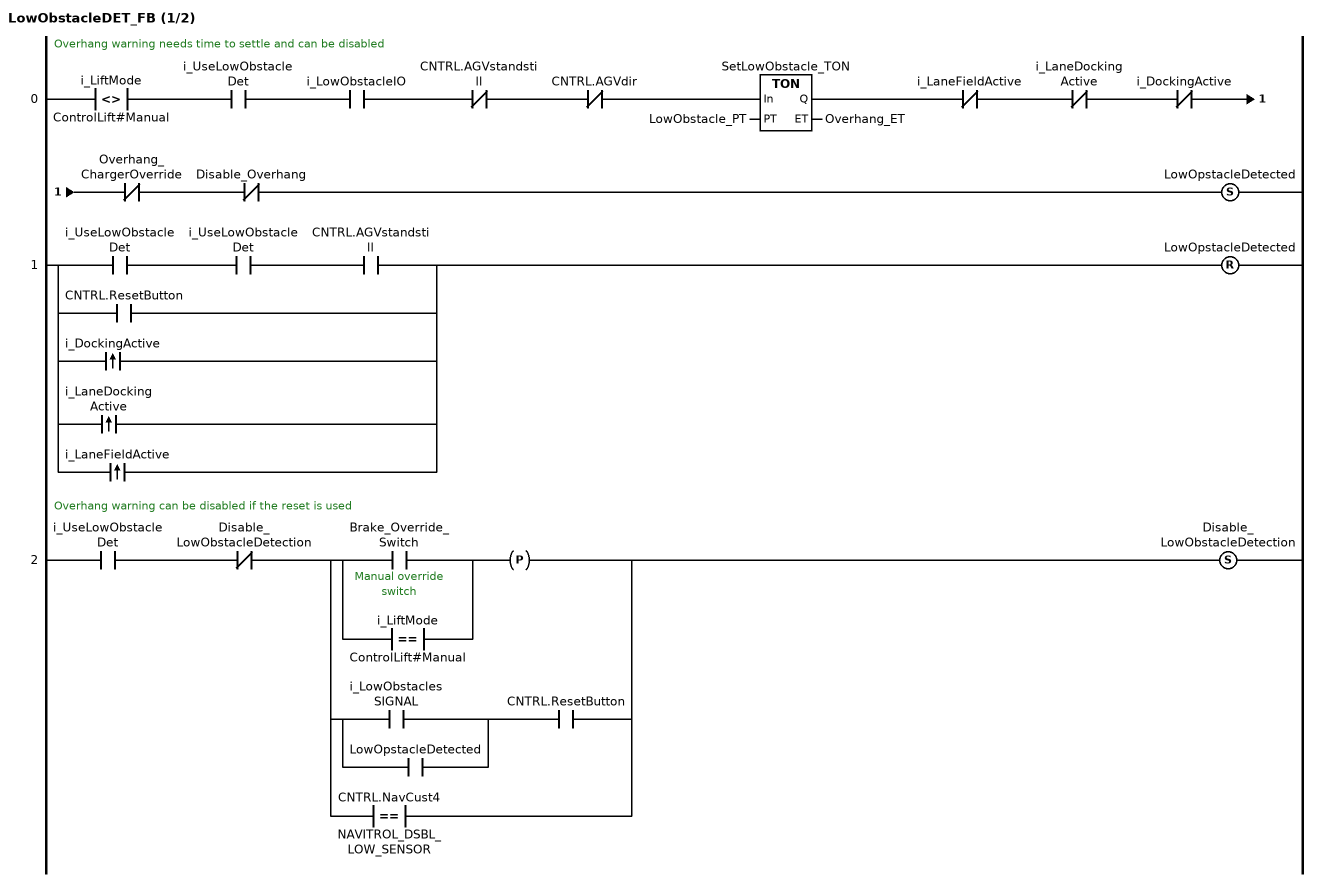
(* Rung 0: Overhang warning needs time to settle and can be disabled *)
SetLowObstacle_TON(In := (i_LiftMode <> ControlLift#Manual) AND i_UseLowObstacleDet AND i_LowObstacleIO AND NOT CNTRL.AGVstandstill AND NOT CNTRL.AGVdir, PT := LowObstacle_PT, ET => Overhang_ET);
IF SetLowObstacle_TON.Q AND NOT i_LaneFieldActive AND NOT i_LaneDockingActive AND NOT i_DockingActive AND NOT Overhang_ChargerOverride AND NOT Disable_Overhang THEN
    LowOpstacleDetected := TRUE;
END_IF;
(* Rung 1 *)
_e1(CLK := i_DockingActive);
_e2(CLK := i_LaneDockingActive);
_e3(CLK := i_LaneFieldActive);
IF (i_UseLowObstacleDet AND i_UseLowObstacleDet AND CNTRL.AGVstandstill) OR CNTRL.ResetButton OR _e1.Q OR _e2.Q OR _e3.Q THEN
    LowOpstacleDetected := FALSE;
END_IF;
(* Rung 2: Overhang warning can be disabled if the reset is used *)
_p4 := i_UseLowObstacleDet AND NOT Disable_LowObstacleDetection;
_e5(CLK := _p4 AND (Brake_Override_Switch OR (i_LiftMode = ControlLift#Manual)));
IF _e5.Q OR (_p4 AND (((i_LowObstaclesSIGNAL OR LowOpstacleDetected) AND CNTRL.ResetButton) OR (CNTRL.NavCust4 = NAVITROL_DSBL_LOW_SENSOR))) THEN
    Disable_LowObstacleDetection := TRUE;
END_IF;

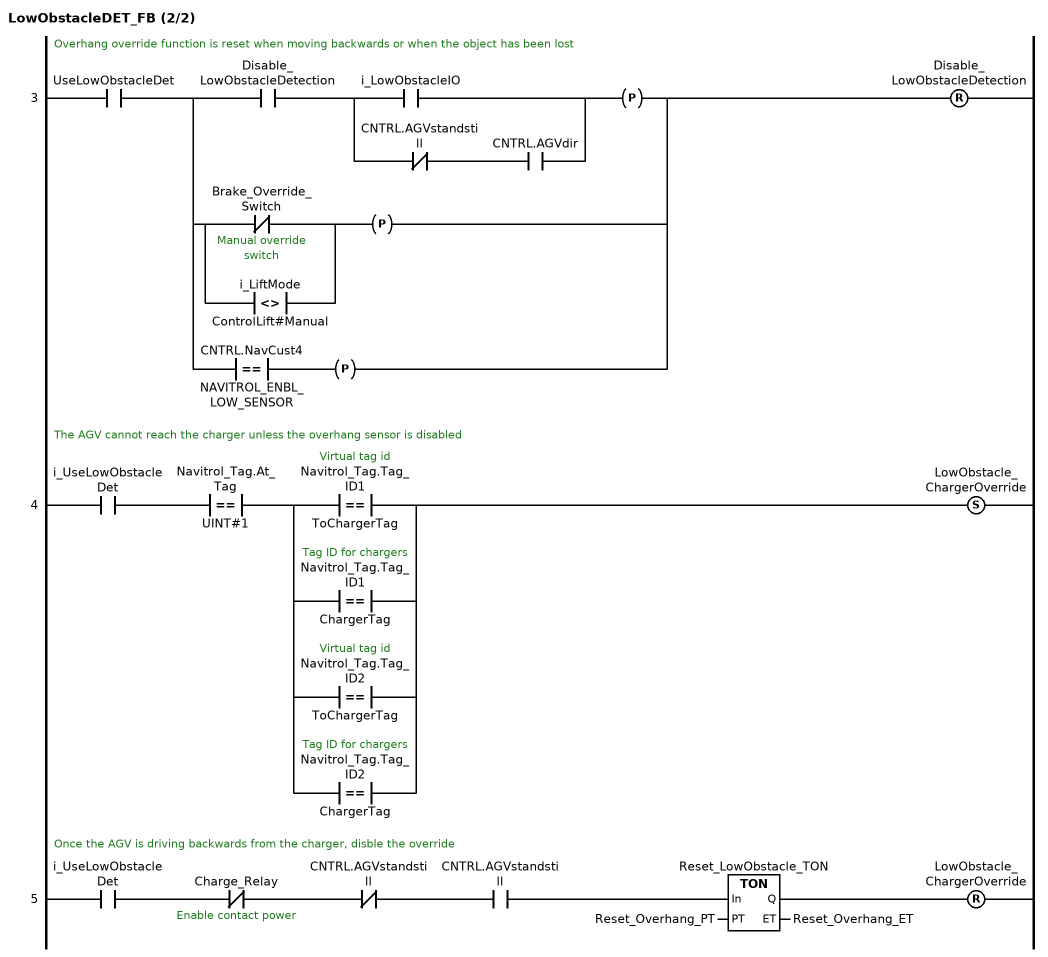
(* Rung 3: Overhang override function is reset when moving backwards or when the object has been lost *)
_e6(CLK := UseLowObstacleDet AND Disable_LowObstacleDetection AND (i_LowObstacleIO OR (NOT CNTRL.AGVstandstill AND CNTRL.AGVdir)));
_e7(CLK := UseLowObstacleDet AND (NOT Brake_Override_Switch OR (i_LiftMode <> ControlLift#Manual)));
_e8(CLK := UseLowObstacleDet AND (CNTRL.NavCust4 = NAVITROL_ENBL_LOW_SENSOR));
IF _e6.Q OR _e7.Q OR _e8.Q THEN Disable_LowObstacleDetection := FALSE; END_IF;
(* Rung 4: The AGV cannot reach the charger unless the overhang sensor is disabled *)
IF i_UseLowObstacleDet AND (Navitrol_Tag.At_Tag = UINT#1) AND ((Navitrol_Tag.Tag_ID1 = ToChargerTag) OR (Navitrol_Tag.Tag_ID1 = ChargerTag) OR (Navitrol_Tag.Tag_ID2 = ToChargerTag) OR (Navitrol_Tag.Tag_ID2 = ChargerTag)) THEN
    LowObstacle_ChargerOverride := TRUE;
END_IF;
(* Rung 5: Once the AGV is driving backwards from the charger, disble the override *)
Reset_LowObstacle_TON(In := i_UseLowObstacleDet AND NOT Charge_Relay AND NOT CNTRL.AGVstandstill AND CNTRL.AGVstandstill, PT := Reset_Overhang_PT, ET => Reset_Overhang_ET);
IF Reset_LowObstacle_TON.Q THEN LowObstacle_ChargerOverride := FALSE; END_IF;
END_FUNCTION_BLOCK

FUNCTION_BLOCK OverhangDET_FB
VAR
    OverhangDetected : BOOL;
    NAVITROL_DISABLE_OVERHANG : REAL := 1;
    NAVITROL_ENABLE_OVERHANG : REAL := 0;
    Disable_Overhang : BOOL;
    Overhang_ChargerOverride : BOOL;
    Overhang_TON : TON;
    Overhang_PT : TIME := T#250ms;
    Overhang_ET : TIME;
    Reset_Overhang_TON : TON;
    Reset_Overhang_PT : TIME := T#1s;
    Reset_Overhang_ET : TIME;
    ReleaseDelay_TON : TON;
    ReleaseDelay_PT : TIME := T#3s;
END_VAR
VAR_INPUT
    ENABLE : BOOL;
    CNTRL : stControl;
    i_DockingActive : BOOL;
    i_LaneFieldActive : BOOL;
    i_LaneDockingActive : BOOL;
    i_Overhang : stOverhang;
    i_LiftMode : ControlLift;
END_VAR
VAR_OUTPUT
    o_OverhangOverruled : BOOL;
    STOP : BOOL;
    ERROR : BOOL;
END_VAR
VAR_EXTERNAL
    Brake_Override_Switch : BOOL;
    Charge_Relay : BOOL;
    Navitrol_Tag : Navitrol_Status_TagV4_sec_struct;
    ToChargerTag : UDINT;
    ChargerTag : UDINT;
END_VAR
VAR
    _e1 : F_TRIG;
    _e2 : F_TRIG;
    _e3 : R_TRIG;
    _e4 : R_TRIG;
    _e5 : R_TRIG;
    _e6 : R_TRIG;
    _e7 : R_TRIG;
    _e8 : F_TRIG;
    _e9 : R_TRIG;
    _e10 : R_TRIG;
    _e11 : R_TRIG;
    _e12 : R_TRIG;
    _e13 : R_TRIG;
    _e14 : R_TRIG;
    _e15 : R_TRIG;
END_VAR
(* ladder, written here as Structured Text *)

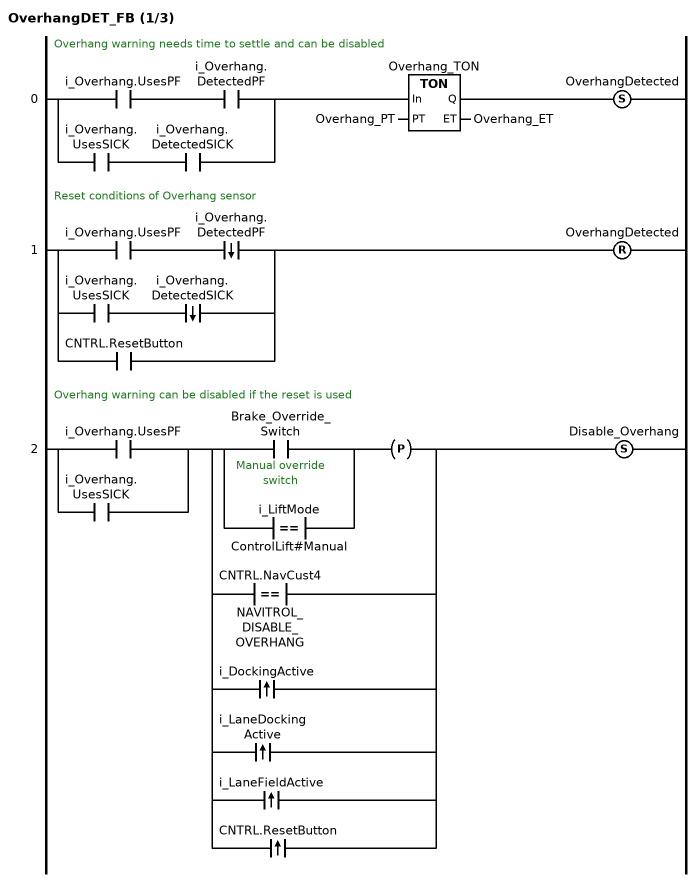
(* Rung 0: Overhang warning needs time to settle and can be disabled *)
Overhang_TON(In := (i_Overhang.UsesPF AND i_Overhang.DetectedPF) OR (i_Overhang.UsesSICK AND i_Overhang.DetectedSICK), PT := Overhang_PT, ET => Overhang_ET);
IF Overhang_TON.Q THEN OverhangDetected := TRUE; END_IF;
(* Rung 1: Reset conditions of Overhang sensor *)
_e1(CLK := i_Overhang.DetectedPF);
_e2(CLK := i_Overhang.DetectedSICK);
IF (i_Overhang.UsesPF AND _e1.Q) OR (i_Overhang.UsesSICK AND _e2.Q) OR CNTRL.ResetButton THEN
    OverhangDetected := FALSE;
END_IF;
(* Rung 2: Overhang warning can be disabled if the reset is used *)
_e3(CLK := (i_Overhang.UsesPF OR i_Overhang.UsesSICK) AND (Brake_Override_Switch OR (i_LiftMode = ControlLift#Manual)));
_e4(CLK := i_DockingActive);
_e5(CLK := i_LaneDockingActive);
_e6(CLK := i_LaneFieldActive);
_e7(CLK := CNTRL.ResetButton);
IF _e3.Q OR ((i_Overhang.UsesPF OR i_Overhang.UsesSICK) AND ((CNTRL.NavCust4 = NAVITROL_DISABLE_OVERHANG) OR _e4.Q OR _e5.Q OR _e6.Q OR _e7.Q)) THEN
    Disable_Overhang := TRUE;
END_IF;

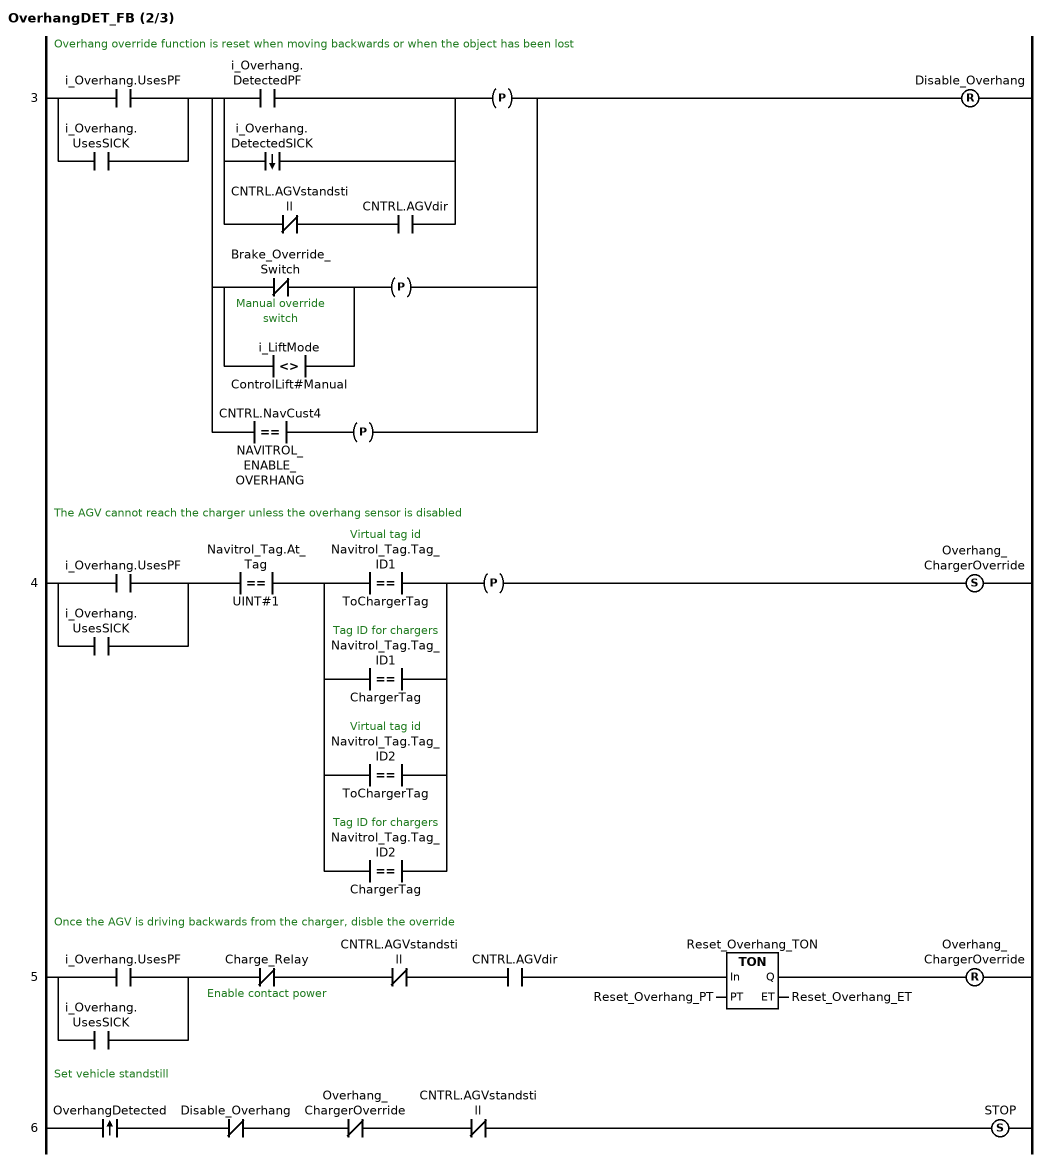
(* Rung 3: Overhang override function is reset when moving backwards or when the object has been lost *)
_e8(CLK := i_Overhang.DetectedSICK);
_e9(CLK := (i_Overhang.UsesPF OR i_Overhang.UsesSICK) AND (i_Overhang.DetectedPF OR _e8.Q OR (NOT CNTRL.AGVstandstill AND CNTRL.AGVdir)));
_e10(CLK := (i_Overhang.UsesPF OR i_Overhang.UsesSICK) AND (NOT Brake_Override_Switch OR (i_LiftMode <> ControlLift#Manual)));
_e11(CLK := (i_Overhang.UsesPF OR i_Overhang.UsesSICK) AND (CNTRL.NavCust4 = NAVITROL_ENABLE_OVERHANG));
IF _e9.Q OR _e10.Q OR _e11.Q THEN Disable_Overhang := FALSE; END_IF;
(* Rung 4: The AGV cannot reach the charger unless the overhang sensor is disabled *)
_e12(CLK := (i_Overhang.UsesPF OR i_Overhang.UsesSICK) AND (Navitrol_Tag.At_Tag = UINT#1) AND ((Navitrol_Tag.Tag_ID1 = ToChargerTag) OR (Navitrol_Tag.Tag_ID1 = ChargerTag) OR (Navitrol_Tag.Tag_ID2 = ToChargerTag) OR (Navitrol_Tag.Tag_ID2 = ChargerTag)));
IF _e12.Q THEN Overhang_ChargerOverride := TRUE; END_IF;
(* Rung 5: Once the AGV is driving backwards from the charger, disble the override *)
Reset_Overhang_TON(In := (i_Overhang.UsesPF OR i_Overhang.UsesSICK) AND NOT Charge_Relay AND NOT CNTRL.AGVstandstill AND CNTRL.AGVdir, PT := Reset_Overhang_PT, ET => Reset_Overhang_ET);
IF Reset_Overhang_TON.Q THEN Overhang_ChargerOverride := FALSE; END_IF;
(* Rung 6: Set vehicle standstill *)
_e13(CLK := OverhangDetected);
IF _e13.Q AND NOT Disable_Overhang AND NOT Overhang_ChargerOverride AND NOT CNTRL.AGVstandstill THEN
    STOP := TRUE;
END_IF;

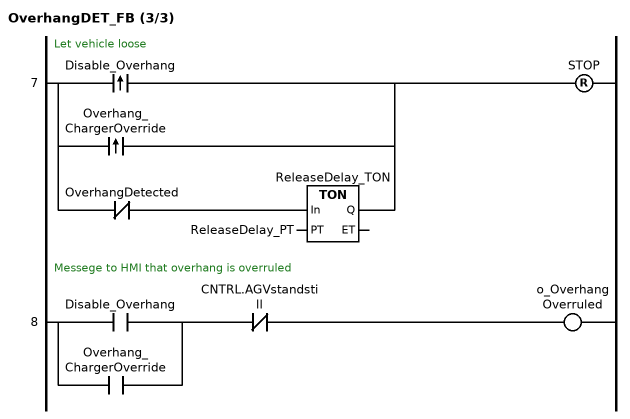
(* Rung 7: Let vehicle loose *)
_e14(CLK := Disable_Overhang);
_e15(CLK := Overhang_ChargerOverride);
ReleaseDelay_TON(In := NOT OverhangDetected, PT := ReleaseDelay_PT);
IF _e14.Q OR _e15.Q OR ReleaseDelay_TON.Q THEN STOP := FALSE; END_IF;
(* Rung 8: Messege to HMI that overhang is overruled *)
o_OverhangOverruled := (Disable_Overhang OR Overhang_ChargerOverride) AND NOT CNTRL.AGVstandstill;
END_FUNCTION_BLOCK